{attribute 'qualified_only'}
{attribute 'strict'}
TYPE eTcoRemoteTaskTests : (
    RestoreTasks := 10,
    InvokeInitializedCSharpMethod := 100,
    InvokeNotInitializedCSharpMethod := 200,
    ExceptionInMethodWillResultInException := 400
);
END_TYPE

(* stored: Version 1.1.0.1
   DUT eTcoRemoteTaskTests: Id {5b47df81-f3f4-0059-0466-9130b7486ad5} *)
